// TIA Portal V16 export
// export: Created 2021-08-30T10:49:35.9355603Z, ExportSetting WithDefaults, DisplayName Totally Integrated Automation Portal, DisplayVersion V16 Update 3, DisplayName TIA Portal Version Control Interface, DisplayVersion V16 Update 2, DisplayName TIA Portal Openness, DisplayVersion V16 Update 3, DisplayName TIA Portal Teamcenter Gateway, DisplayVersion V16, DisplayName STEP 7 Professional, DisplayVersion V16 Update 3, DisplayName STEP 7 Safety, DisplayVersion V16, DisplayName WinCC Advanced, DisplayVersion V16 Update 3
VAR_GLOBAL   // PLC tag table "A1_DI"
   iP301_Run AT %I0.0 : Bool;   // P301 Робота
   iP302_Run AT %I0.1 : Bool;   // P302 Робота
   iP1201_Run AT %I0.2 : Bool;   // P1201 Робота
   iP1202_Run AT %I0.3 : Bool;   // P1202 Робота
   iP1501_Run AT %I0.4 : Bool;   // P1501 Робота
   iP1502_Run AT %I0.5 : Bool;   // P1502 Робота
   iP70x_Ready AT %I0.6 : Bool;   // P70x Готовність
   iP701_Run AT %I0.7 : Bool;   // P701 Робота
   iP702_Run AT %I1.0 : Bool;   // P702 Робота
   iP201_Ready AT %I1.1 : Bool;   // P201 Готовність
   iP201_Run AT %I1.2 : Bool;   // P201 Робота
   iC501_Ready AT %I1.3 : Bool;   // C501 Готовність
   iStop AT %I1.4 : Bool;   // Аварійне вимикання
   iSF_Fail AT %I1.5 : Bool;   // Аварія захисних автоматів
END_VAR
VAR_GLOBAL CONSTANT   // user constants
   "iP-301_Run" : Int := 0;
   "iP-302_Run" : Int := 1;
   "iP-1201_Run" : Int := 2;
   "iP-1202_Run" : Int := 3;
   "iP-1501_Run" : Int := 4;
   "iP-1502_Run" : Int := 5;
   "iP-70x_Ready" : Int := 6;
   "iP-701_Run" : Int := 7;
   "iP-702_Run" : Int := 8;
   "iP-201_Ready" : Int := 9;
   "iP-201_Run" : Int := 10;
   "iC-501_Ready" : Int := 11;
   i_Stop : Int := 12;
   i_SF_Fail : Int := 13;
END_VAR
